Fanuc KAREL source: kt00479.KL

-- PROVISIONAL review KL for V770-1; original PC SHA256 7e264e44622a4ea422c2591a0e1fd4f1a17716f7b1c9b8512df04950aa0247d6
-- Incomplete behavior may be omitted. Consult companion uncertainty JSON. Do not deploy.
PROGRAM KT00479
%NOLOCKGROUP
-- UNRESOLVED_DECL P1 type=000101
-- UNRESOLVED_DECL P2 type=000102
-- UNRESOLVED_DECL OUT type=000101
BEGIN
  -- UNRESOLVED_PC offsets 5-20; opcodes 2E,22,32,35
  -- UNRESOLVED_PC offsets 25-54; opcodes 49,49,7E,60,4A
  -- UNRESOLVED_PC offsets 59-63; opcodes 7F
END KT00479
